{attribute 'GeneratedUsingTerminal: EJ7342-0000-0019'}
{attribute addProperty BoxType "EJ7342-0000-0019"}
{attribute addProperty Id "StatusAT %I*Status_3035BE2E10Counter_valueAT %I*UINT2Latch_valueAT %I*UINT2"}
{attribute addProperty CRC "3696597680"}
{attribute addProperty Size "14"}
TYPE ENC_Status_compact_Channel_DC559AB0 EXTENDS InputBase_8311D824 :
STRUCT
	{attribute addProperty Name "Status"}
	Status AT %I* : Status_3035BE2E;
	{attribute addProperty Name "Counter_value"}
	Counter_value AT %I* : UINT;
	{attribute addProperty Name "Latch_value"}
	Latch_value AT %I* : UINT;
END_STRUCT
END_TYPE

(* stored: Version 1.2.0.0, ProductVersion 3.1.4024.9
   DUT ENC_Status_compact_Channel_DC559AB0: Id {1feb74c6-c1c4-42d8-a7f7-7c354886520e} *)
